// TIA Portal V16 export
// export: Created 2022-06-11T10:19:43.3098556Z, ExportSetting WithDefaults, DisplayName Totally Integrated Automation Portal, DisplayVersion V16 Update 3, DisplayName TIA Portal Version Control Interface, DisplayVersion V16 Update 2, DisplayName TIA Portal Openness, DisplayVersion V16 Update 3, DisplayName STEP 7 Professional, DisplayVersion V16 Update 3, DisplayName STEP 7 Safety, DisplayVersion V16, DisplayName WinCC Professional, DisplayVersion V16 Update 3
DATA_BLOCK "DB11011_St_DevValve3Way"   // DB11011
TITLE = Static DB [DEVICE DRIVER] — Three-Way Valve
{ S7_Optimized_Access := 'TRUE' }
AUTHOR : M_Gledhill
FAMILY : DeviceDriver
NAME : St_DevValve3Way
VERSION : 0.8
// PRACTICAL SERIES AUTOMATION LIBRARY (PAL)   —   COPYRIGHT 2020 – M. GLEDHILL (MIT LICENCE)
//                   ———— ◆ ————
// FULL ONLINE DOCUMENTATION IS AVAILABLE AT: https://practicalseries.com/2001-pal/index.html
// stored: AutoNumber false, DBAccessibleFromOPCUA true, IsOnlyStoredInLoadMemory false, IsRetainMemResEnabled false, IsWriteProtectedInAS false, MemoryReserve 100
   VAR
      _DB_Header { ExternalAccessible := 'False'; ExternalVisible := 'False'; ExternalWritable := 'False'} : Array[0..79] of Bool;   // Static DB [DEVICE DRIVER] — Three-way Valve
      __________0000_0 { ExternalAccessible := 'False'; ExternalVisible := 'False'; ExternalWritable := 'False'} : Bool := false;
      __________0000_1 { ExternalAccessible := 'False'; ExternalVisible := 'False'; ExternalWritable := 'False'} : Bool := false;   // ▀▀▀▀ DB CURRENT REVISION
      revInfo { ExternalWritable := 'False'; S7_SetPoint := 'True'} : "UT01000_St_SysRevision";   // Revision information
      __________0010_0 { ExternalAccessible := 'False'; ExternalVisible := 'False'; ExternalWritable := 'False'} : Bool := false;
      __________0010_1 { ExternalAccessible := 'False'; ExternalVisible := 'False'; ExternalWritable := 'False'} : Bool := false;   // ▀▀▀▀ THREE-WAY VALVES
      V001 { ExternalWritable := 'False'; S7_SetPoint := 'True'} : "UT11011_St_DevValve3Way";   // Filter 1 backwash divert
   END_VAR
BEGIN
   // _DB_Header[0] : ▄▄▄▄▄▄▄▄▄▄▄▄▄▄▄▄▄▄▄▄▄▄▄▄▄▄▄▄▄▄▄▄▄ ＳＴＡＮＤＡＲＤ ▄▄
   // _DB_Header[2] : TITLE: DEVICE DRIVER — THREE-WAY VALVE
   // _DB_Header[4] : ▀▀▀▀▀▀▀▀▀▀▀▀▀▀▀▀▀▀▀▀▀▀▀▀▀▀▀▀▀▀▀▀▀▀▀▀▀▀▀▀▀▀▀▀
   // _DB_Header[5] : TYPE: STATIC
   // _DB_Header[6] : ▄▄▄▄▄▄▄▄▄▄▄▄▄▄▄▄▄▄▄▄▄▄▄▄▄▄▄▄▄▄▄▄▄▄▄▄▄▄▄▄▄▄▄▄
   // _DB_Header[8] : This is the static data block associated with the standard device driver for a three-way valve
   // _DB_Header[9] : block:
   // _DB_Header[10] : FC11011_StdDevValve3Way
   // _DB_Header[12] : The static data holds the configuration data for the device ( limit switch and
   // _DB_Header[13] : interlock configuration &c.)
   // _DB_Header[15] : Each valve is given the user data type:
   // _DB_Header[16] : UT11011_St_DevValve3Way
   // _DB_Header[17] : This holds the full set of static configuration data for the device
   // _DB_Header[19] : ━━━ ⬙⬙⬙⬙⬙⬙ ━━━
   // _DB_Header[21] : ▄▄▄▄▄▄▄▄▄▄▄▄▄▄▄▄▄▄▄▄▄▄▄▄▄▄▄▄▄▄▄▄▄▄▄▄▄▄▄▄▄▄▄▄
   // _DB_Header[22] : MODIFICATION HISTORY
   // _DB_Header[24] : This is a summary of the recent software modifications made to this block (most recent at top)
   // _DB_Header[26] : ―――――――――――――――――――――――――――――――――――――――――――
   // _DB_Header[27] : DATE REVISION MASTER BRANCH DEV
   // _DB_Header[28] : (nnn.amm) COMMIT TAG (Base ---> Merge) BRANCH Author
   // _DB_Header[29] : ———————————————————————————————————————————
   // _DB_Header[30] : 2022.06.07 000.801 D0014A-000.801 D0014 N/A D0014A M. Gledhill
   // _DB_Header[31] : Released for test (SMTS)
   // _DB_Header[33] : 2022.06.01 000.101 D0014A-000.101 D0014 N/A D0014A M. Gledhill
   // _DB_Header[34] : FC11011 Block created
   // _DB_Header[35] : ———————————————————————————————————————————
   // _DB_Header[36] : Where: nnn = Major revision
   // _DB_Header[37] : a = Type (1-7 Development, 8 Proving, 9 Qualification, 0 Release)
   // _DB_Header[38] : mm = Minor revision (must be 00 if a = 0)
   // _DB_Header[39] : Block properties version number should be set to nn.a (only one decimal place)
   // _DB_Header[41] : ██████████████ █ █ █ █ END █ █ █ █ ██████████████
   revInfo.REV_BLOCK := 'DB11011';
   revInfo.REV_NUMBER := '000.801';
   revInfo.REV_DATE := '2022.06.07';
   revInfo.REV_AUTHOR := 'M. Gledhill';
   V001.CONFIG_FBK_ENG_EN := true;
   V001.CONFIG_FBK_DENG_EN := true;
   V001.INFO_TAG := 'V001';
   V001.TIME_ENG_MAX := 20.0;
   V001.TIME_DENG_MAX := 30.0;
   V001.TIME_DER_ENG := 80.0;
   V001.TIME_DER_DENG := 90.0;
END_DATA_BLOCK
